TYPE ST_SheepingPictureFeeback :
STRUCT
	CameraPositionDone : BOOL;
END_STRUCT
END_TYPE

(* stored: Version 1.1.0.1, ProductVersion 3.1.4024.13
   DUT ST_SheepingPictureFeeback: Id {94241eaa-0f4e-4e91-a6c0-47309d572fe6} *)
